PROGRAM Axis04_Auto
VAR
	Always_ON	:	BOOL	:=TRUE	;//상시 ON 
	Always_OFF	:	BOOL	:=FALSE	;//상시 OFF
END_VAR

// NETWORK 1

END_PROGRAM

(* stored: Version 1.1.0.1, ProductVersion 3.1.4024.15
   POU Axis04_Auto: Id {0735a1ba-c4fd-4580-8e71-47f2213f5fd9}, SpecialFunc None *)
